{attribute addProperty BoxType "EK1122-0000-0018"}
{attribute addProperty Id "Beckhoff_ER6xxxsub_EK1100EK1100_179A0949162A_0001_ER6001_0002_0016ER6001_7904467646658.25A_0002_ER6001_0002_0021ER6001_7904467646658.25A_0003_ER6002_0002_0021ER6002_320F021A850106.25A_0004_ER6002_0002_0022ER6002_FC20A988850106.25A_0005_ER6002_0002_0023ER6002_FC20A988850106.25"}
{attribute addProperty CRC "2127943795"}
{attribute addProperty SizeInBites "3498"}
{attribute addProperty SizeInBytes "437.25"}
TYPE Beckhoff_ER6xxxEK1122_7ED5D873 EXTENDS EK1122_179A0949 :
STRUCT
	{attribute addProperty Name "Beckhoff_ER6xxxsub_EK1100"}
	Beckhoff_ER6xxxsub_EK1100 : EK1100_179A0949;
	{attribute addProperty Name "A_0001_ER6001_0002_0016"}
	A_0001_ER6001_0002_0016 : ER6001_79044676;
	{attribute addProperty Name "A_0002_ER6001_0002_0021"}
	A_0002_ER6001_0002_0021 : ER6001_79044676;
	{attribute addProperty Name "A_0003_ER6002_0002_0021"}
	A_0003_ER6002_0002_0021 : ER6002_320F021A;
	{attribute addProperty Name "A_0004_ER6002_0002_0022"}
	A_0004_ER6002_0002_0022 : ER6002_FC20A988;
	{attribute addProperty Name "A_0005_ER6002_0002_0023"}
	A_0005_ER6002_0002_0023 : ER6002_FC20A988;
END_STRUCT
END_TYPE

(* stored: Version 1.2.0.0, ProductVersion 3.1.4024.9
   DUT Beckhoff_ER6xxxEK1122_7ED5D873: Id {b997a9dc-743f-48f7-9c2a-744113c3830c} *)
